VAR_GLOBAL
	fbMachineTime : FB_LocalSystemTime;
	fbMachineLogger : FB_FileLogger;
END_VAR

(* stored: Version 1.1.0.1, ProductVersion 3.1.4024.12
   GVL GVL: Id {6ede5a0f-6838-4c0f-a067-40155c90d7a1} *)
